(*********************************** G.D S.p.A. - Technical Department ***********************************
============= PROGRAM INFO ============
FOLDER:             TBD
MACHINES INVOLVED:  TBD 

============= DESCRIPTION =============
csp main interface program

============= REVISIONS ===============
Date		Version	 	Author      	Description             
----------	-------		------------  	--------------------------------------------
2019/09/27 	0000.00	 	M.Grasso		Creation of the PRG

**********************************************************************************************************)
PROGRAM _csp_transfer_upstacker_low
VAR
END_VAR

(* TRANSFER *)
	(* UPSTACKER *)
		(* BACKSTOP *)
		;
		(* BELT *)
		;
		(* DOWNSTREAM *)
		;
		(* SENSORS *)
		;
		(* UPSTREAM *)
		;

END_PROGRAM

(* stored: Version 1.1.0.1, ProductVersion 3.1.4022.9
   POU _csp_transfer_upstacker_low: Id {8183ced4-c691-40b8-903f-8eba41e82476}, SpecialFunc None *)
